// TIA Portal V20 export
TYPE "type_emRelations_em9_sequence"
// stored: Access Published, Namespace Unit1
   STRUCT
      vision : Struct
         jobs : "LAF_typeJobs";
         sequence : "LAF_typeSequence";
         selectJobStatus { S7_SetPoint := 'True'} : Array[0..10] of "LAF_typeJobStatus";
         "step" : "LER_typeStep";
         jobInterface : Struct
            loadJob2 : "LER_typeJobInterface";
            inspectionJob3 : "LER_typeJobInterface";
            unloadJob4 : "LER_typeJobInterface";
         END_STRUCT;
         homeCheck : Struct
            liftDownLightUpPartNoDetect { ExternalWritable := 'False'} : Bool;
            liftDownLightUpPartDetect { ExternalWritable := 'False'} : Bool;
            liftDownLightDownPartDetect { ExternalWritable := 'False'} : Bool;
            liftUpLightUp { ExternalWritable := 'False'} : Bool;
         END_STRUCT;
      END_STRUCT;
      GaugeRnR_Vision : Struct
         jobs : "LAF_typeJobs";
         sequence : "LAF_typeSequence";
         selectJobStatus { S7_SetPoint := 'True'} : Array[0..10] of "LAF_typeJobStatus";
         "step" : "LER_typeStep";
         jobInterface : Struct
            loadJob2 : "LER_typeJobInterface";
            inspectionJob3 : "LER_typeJobInterface";
            unloadJob4 : "LER_typeJobInterface";
         END_STRUCT;
      END_STRUCT;
   END_STRUCT;
   // // vision."step".action1[101] : Step[101] : JOB[1] Condition
   // // vision."step".action1[110] : Step[110] : Light Up
   // // vision."step".action1[130] : Step[130] : Stage Lift Up
   // // vision."step".action1[140] : Step[140] : Hot Press Right JR Detection Check
   // // vision."step".action1[141] : Step[141] : Hot Press Right JR Detection Check Completed
   // // vision."step".action1[160] : Step[160] : Stage Lift Down
   // // vision."step".action1[190] : Step[190] : JOB[1] Step End
   // // vision."step".action1[201] : Step[201] : JOB[2] Condition
   // // vision."step".action1[210] : Step[210] : Vision Loading Request => Transfer PP Right
   // // vision."step".action1[230] : Step[230] : Stage Lift Up
   // // vision."step".action1[240] : Step[240] : Vision Loading Check => Transfer PP Right
   // // vision."step".action1[290] : Step[290] : JOB[2] Step End
   // // vision."step".action1[301] : Step[301] : JOB[3] Condition
   // // vision."step".action1[310] : Step[310] : Stage Lift Down
   // // vision."step".action1[311] : Step[311] : Stage JR Detection Check
   // // vision."step".action1[320] : Step[320] : Light Down
   // // vision."step".action1[330] : Step[330] : Vision Start
   // // vision."step".action1[331] : Step[331] : Vision Result
   // // vision."step".action1[390] : Step[390] : JOB[3] Step End
   // // vision."step".action1[401] : Step[401] : JOB[4] Condition
   // // vision."step".action1[410] : Step[410] : Light Up
   // // vision."step".action1[420] : Step[420] : Stage Lift Up
   // // vision."step".action1[430] : Step[430] : Vision Unloading Request => Transfer PP Right
   // // vision."step".action1[431] : Step[431] : Vision Unloading Check => Transfer PP Right
   // // vision."step".action1[480] : Step[480] : Stage Lift Down
   // // vision."step".action1[490] : Step[490] : JOB[4] Step End
   // // vision."step".transition1[101] : Step[101] : JOB[1] Condition
   // // vision."step".transition1[110] : Step[110] : Light Up
   // // vision."step".transition1[130] : Step[130] : Stage Lift Up
   // // vision."step".transition1[140] : Step[140] : Hot Press Right JR Detection Check
   // // vision."step".transition1[141] : Step[141] : Hot Press Right JR Detection Check Completed
   // // vision."step".transition1[160] : Step[160] : Stage Lift Down
   // // vision."step".transition1[190] : Step[190] : JOB[1] Step End
   // // vision."step".transition1[201] : Step[201] : JOB[2] Condition
   // // vision."step".transition1[210] : Step[210] : Vision Loading Request => Transfer PP Right
   // // vision."step".transition1[230] : Step[230] : Stage Lift Up
   // // vision."step".transition1[240] : Step[240] : Vision Loading Check => Transfer PP Right
   // // vision."step".transition1[290] : Step[290] : JOB[2] Step End
   // // vision."step".transition1[301] : Step[301] : JOB[3] Condition
   // // vision."step".transition1[310] : Step[310] : Stage Lift Down
   // // vision."step".transition1[311] : Step[311] : Stage JR Detection Check
   // // vision."step".transition1[320] : Step[320] : Light Down
   // // vision."step".transition1[330] : Step[330] : Vision Start
   // // vision."step".transition1[331] : Step[331] : Vision Result
   // // vision."step".transition1[390] : Step[390] : JOB[3] Step End
   // // vision."step".transition1[401] : Step[401] : JOB[4] Condition
   // // vision."step".transition1[410] : Step[410] : Light Up
   // // vision."step".transition1[420] : Step[420] : Stage Lift Up
   // // vision."step".transition1[430] : Step[430] : Vision Unloading Request => Transfer PP Right
   // // vision."step".transition1[431] : Step[431] : Vision Unloading Check => Transfer PP Right
   // // vision."step".transition1[480] : Step[480] : Stage Lift Down
   // // vision."step".transition1[490] : Step[490] : JOB[4] Step End
   // // GaugeRnR_Vision."step".action1[101] : Step[101] : JOB[1] Condition
   // // GaugeRnR_Vision."step".action1[110] : Step[110] : Light Up
   // // GaugeRnR_Vision."step".action1[130] : Step[130] : Stage Lift Up
   // // GaugeRnR_Vision."step".action1[140] : Step[140] : Hot Press Right JR Detection Check
   // // GaugeRnR_Vision."step".action1[141] : Step[141] : Hot Press Right JR Detection Check Completed
   // // GaugeRnR_Vision."step".action1[160] : Step[160] : Stage Lift Down
   // // GaugeRnR_Vision."step".action1[190] : Step[190] : JOB[1] Step End
   // // GaugeRnR_Vision."step".action1[201] : Step[201] : JOB[2] Condition
   // // GaugeRnR_Vision."step".action1[210] : Step[210] : Vision Loading Request => Transfer PP Right
   // // GaugeRnR_Vision."step".action1[230] : Step[230] : Stage Lift Up
   // // GaugeRnR_Vision."step".action1[240] : Step[240] : Vision Loading Check => Transfer PP Right
   // // GaugeRnR_Vision."step".action1[290] : Step[290] : JOB[2] Step End
   // // GaugeRnR_Vision."step".action1[301] : Step[301] : JOB[3] Condition
   // // GaugeRnR_Vision."step".action1[310] : Step[310] : Stage Lift Down
   // // GaugeRnR_Vision."step".action1[311] : Step[311] : Stage JR Detection Check
   // // GaugeRnR_Vision."step".action1[320] : Step[320] : Light Down
   // // GaugeRnR_Vision."step".action1[330] : Step[330] : Vision Start
   // // GaugeRnR_Vision."step".action1[331] : Step[331] : Vision Result
   // // GaugeRnR_Vision."step".action1[390] : Step[390] : JOB[3] Step End
   // // GaugeRnR_Vision."step".action1[401] : Step[401] : JOB[4] Condition
   // // GaugeRnR_Vision."step".action1[410] : Step[410] : Light Up
   // // GaugeRnR_Vision."step".action1[420] : Step[420] : Stage Lift Up
   // // GaugeRnR_Vision."step".action1[430] : Step[430] : Vision Unloading Request => Transfer PP Right
   // // GaugeRnR_Vision."step".action1[431] : Step[431] : Vision Unloading Check => Transfer PP Right
   // // GaugeRnR_Vision."step".action1[480] : Step[480] : Stage Lift Down
   // // GaugeRnR_Vision."step".action1[490] : Step[490] : JOB[4] Step End
   // // GaugeRnR_Vision."step".transition1[101] : Step[101] : JOB[1] Condition
   // // GaugeRnR_Vision."step".transition1[110] : Step[110] : Light Up
   // // GaugeRnR_Vision."step".transition1[130] : Step[130] : Stage Lift Up
   // // GaugeRnR_Vision."step".transition1[140] : Step[140] : Hot Press Right JR Detection Check
   // // GaugeRnR_Vision."step".transition1[141] : Step[141] : Hot Press Right JR Detection Check Completed
   // // GaugeRnR_Vision."step".transition1[160] : Step[160] : Stage Lift Down
   // // GaugeRnR_Vision."step".transition1[190] : Step[190] : JOB[1] Step End
   // // GaugeRnR_Vision."step".transition1[201] : Step[201] : JOB[2] Condition
   // // GaugeRnR_Vision."step".transition1[210] : Step[210] : Vision Loading Request => Transfer PP Right
   // // GaugeRnR_Vision."step".transition1[230] : Step[230] : Stage Lift Up
   // // GaugeRnR_Vision."step".transition1[240] : Step[240] : Vision Loading Check => Transfer PP Right
   // // GaugeRnR_Vision."step".transition1[290] : Step[290] : JOB[2] Step End
   // // GaugeRnR_Vision."step".transition1[301] : Step[301] : JOB[3] Condition
   // // GaugeRnR_Vision."step".transition1[310] : Step[310] : Stage Lift Down
   // // GaugeRnR_Vision."step".transition1[311] : Step[311] : Stage JR Detection Check
   // // GaugeRnR_Vision."step".transition1[320] : Step[320] : Light Down
   // // GaugeRnR_Vision."step".transition1[330] : Step[330] : Vision Start
   // // GaugeRnR_Vision."step".transition1[331] : Step[331] : Vision Result
   // // GaugeRnR_Vision."step".transition1[390] : Step[390] : JOB[3] Step End
   // // GaugeRnR_Vision."step".transition1[401] : Step[401] : JOB[4] Condition
   // // GaugeRnR_Vision."step".transition1[410] : Step[410] : Light Up
   // // GaugeRnR_Vision."step".transition1[420] : Step[420] : Stage Lift Up
   // // GaugeRnR_Vision."step".transition1[430] : Step[430] : Vision Unloading Request => Transfer PP Right
   // // GaugeRnR_Vision."step".transition1[431] : Step[431] : Vision Unloading Check => Transfer PP Right
   // // GaugeRnR_Vision."step".transition1[480] : Step[480] : Stage Lift Down
   // // GaugeRnR_Vision."step".transition1[490] : Step[490] : JOB[4] Step End
END_TYPE
